{attribute 'qualified_only'}
VAR_GLOBAL
    // 与外部Python Vision Service通过ADS交换的唯一同轴度视觉接口。
    stInterface : ST_CoaxVisionInterface;
END_VAR

(* stored: Version 1.1.0.1, ProductVersion 3.1.4026.20
   GVL GVL_CoaxVision: Id {074C5908-93CB-4DD5-9BC0-C5CD05653C1C} *)
